Yaskawa INFORM job: HOME_POS.JBI

/JOB
//NAME HOME_POS
//POS
///NPOS 0,0,0,4,0,0
///TOOL 0
///POSTYPE ROBOT
///RECTAN
///RCONF 0,0,0,0,0,0,0,0,0,0,0,0,0,0,0,0,0,0,0,0,0,0,0,0
P00000=10.000,0.000,0.000,0.0000,0.0000,0.0000
///POSTYPE BASE
P00001=249,16.200,273.300,-179.4000,-0.79,-160.6000
//INST
///DATE 2017/03/31 08:11
///ATTR SC,RW
///GROUP1 RB1
NOP
MOVL P00001 V=50 NWAIT ACC=100 DEC=100
END
